INTERFACE I_Resettable

METHOD PUBLIC Reset : HRESULT
VAR_INPUT
END_VAR
END_METHOD

END_INTERFACE

(* stored: Version 1.1.0.1
   Itf I_Resettable: Id {9dcd830e-9ab4-4ce2-a3e2-d2a7698b4f77}
   Method Reset: Id {98586d87-7191-416b-9787-61b6e82fe760} *)
